// TwinCAT 3 PLC project Assembly_2_PLC
// ProgramVersion: 3.1.4022.7
// libraries:
//   Tc2_Standard, * (Beckhoff Automation GmbH)
//   Tc2_System, * (Beckhoff Automation GmbH)
//   Tc3_Module, * (Beckhoff Automation GmbH)
// project tree:
//   GVLs/ HMI.TcGVL
//   / PlcTask.TcTTO
//   POUs/00 System/ fbControl.TcPOU
//   POUs/01 Infeed/ fbInConveyor.TcPOU
//   POUs/02 Fitting/ fbHousingDelivery.TcPOU, fbInsertPlacing.TcPOU
//   POUs/03 Pressing/ fbHandling.TcPOU, fbPressing.TcPOU
//   POUs/ MAIN.TcPOU
// real-time tasks:
//   TASK PlcTask: cycle T#10ms, priority 20, ADS port 350
// I/O:
//   DEVICE Device 2 (EtherCAT), AmsNetId 10.133.61.48.3.1
//     Term 1 (EK1814) Console [EK1814 EtherCAT IO-Coupler  (0,5A E-Bus, 4 Ch. Dig. In, 3ms, 4 Ch. Dig. Out 24V, 0,5A)]
//       Term 2 (EL6900) FS Logic [EL6900, TwinSAFE PLC]
//       Term 3 (EL1904) FS DI1 [EL1904, 4 Ch. Safety Input 24V, TwinSAFE]
//         modules: Module 1 (FSOES)
//       Term 4 (EL1904) FS DI2 [EL1904, 4 Ch. Safety Input 24V, TwinSAFE]
//         modules: Module 1 (FSOES)
//       Term 5 (EL2904) FS DQ [EL2904, 4 Ch. Safety Output 24V, 0.5A, TwinSAFE]
//         modules: Module 1 (FSOES), Module 2 (DO)
//       Term 6 (EL1809) ST DI [EL1809 16Ch. Dig. Input 24V, 3ms]
//       Term 7 (EL2809) ST DQ [EL2809 16Ch. Dig. Output 24V, 0.5A]
//       Term 8 (EK1110) [EK1110 EtherCAT extension]
//     Term 9 (EK1100) Placing [EK1100 EtherCAT Coupler (2A E-Bus)]
//       Term 10 (EL1809) ST DI [EL1809 16Ch. Dig. Input 24V, 3ms]
//       Term 11 (EL2809) ST DQ [EL2809 16Ch. Dig. Output 24V, 0.5A]
//       Term 23 (EL9011) [EL9011 End Terminal]
//     Term 12 (EK1100) Pressing [EK1100 EtherCAT Coupler (2A E-Bus)]
//       Term 13 (EL1809) ST DI [EL1809 16Ch. Dig. Input 24V, 3ms]
//       Term 14 (EL2809) ST DQ [EL2809 16Ch. Dig. Output 24V, 0.5A]
//       Term 15 (EL3102) ST AI [EL3102 2Ch. Ana. Input +/-10V, Diff.]
//       Term 16 (EL4032) ST AQ [EL4032 2Ch. Ana. Output +/-10V, 12bit]
//       Term 24 (EL9011) [EL9011 End Terminal]
//     Term 17 (EK1100) External [EK1100 EtherCAT Coupler (2A E-Bus)]
//       Term 18 (EL1904) FS DI1 [EL1904, 4 Ch. Safety Input 24V, TwinSAFE]
//         modules: Module 1 (FSOES)
//       Term 19 (EL1904) FS DI2 [EL1904, 4 Ch. Safety Input 24V, TwinSAFE]
//         modules: Module 1 (FSOES)
//       Term 20 (EL2904) FS DQ [EL2904, 4 Ch. Safety Output 24V, 0.5A, TwinSAFE]
//         modules: Module 1 (FSOES), Module 2 (DO)
//       Term 21 (EL1808) ST DI [EL1808 8Ch. Dig. Input 24V, 3ms]
//       Term 22 (EL2808) ST DQ [EL2808 8Ch. Dig. Output 24V, 0.5A]
//       Term 25 (EL9011) [EL9011 End Terminal]
// variable links:
//   Device 2 (EtherCAT) <-> Device 2 (EtherCAT)/Term 1 (EK1814) Console/Term 2 (EL6900) FS Logic
//     Term 1 (EK1814) Console/Term 3 (EL1904) FS DI1/Module 1 (FSOES)/RxPDO/FSOE <-> ConnectionInputs/Message_2 TxPDO
//     Term 1 (EK1814) Console/Term 3 (EL1904) FS DI1/Module 1 (FSOES)/TxPDO/FSOE <-> ConnectionOutputs/Message_2 RxPDO
//     Term 1 (EK1814) Console/Term 5 (EL2904) FS DQ/Module 1 (FSOES)/TxPDO/FSOE <-> ConnectionOutputs/Message_4 RxPDO
//     Term 17 (EK1100) External/Term 20 (EL2904) FS DQ/Module 1 (FSOES)/RxPDO/FSOE <-> ConnectionInputs/Message_7 TxPDO
//     Term 17 (EK1100) External/Term 20 (EL2904) FS DQ/Module 1 (FSOES)/TxPDO/FSOE <-> ConnectionOutputs/Message_7 RxPDO
//   Device 2 (EtherCAT) <-> Device 2 (EtherCAT)/Term 1 (EK1814) Console/Term 4 (EL1904) FS DI2
//     Term 1 (EK1814) Console/Term 2 (EL6900) FS Logic/ConnectionInputs/Message_3 TxPDO <-> Module 1 (FSOES)/RxPDO/FSOE
//     Term 1 (EK1814) Console/Term 2 (EL6900) FS Logic/ConnectionOutputs/Message_3 RxPDO <-> Module 1 (FSOES)/TxPDO/FSOE
//   Device 2 (EtherCAT) <-> Device 2 (EtherCAT)/Term 1 (EK1814) Console/Term 5 (EL2904) FS DQ
//     Term 1 (EK1814) Console/Term 2 (EL6900) FS Logic/ConnectionInputs/Message_4 TxPDO <-> Module 1 (FSOES)/RxPDO/FSOE
//   Assembly_2_PLC/Assembly_2_PLC Instance <-> Device 2 (EtherCAT)/Term 1 (EK1814) Console/Term 2 (EL6900) FS Logic
//     PlcTask Inputs/MAIN.estopPressed <-> StandardInputs/Standard Out Var 9
//     PlcTask Inputs/MAIN.systemOk <-> StandardInputs/Standard Out Var 10
//     PlcTask Outputs/MAIN.doorUnlock_But <-> StandardOutputs/Standard In Var 8
//     PlcTask Outputs/MAIN.safeGroupErrorReset <-> StandardOutputs/Standard In Var 1

CONFIGURATION Assembly_2_PLC
    RESOURCE PLC ON TwinCAT3
        TASK PlcTask(INTERVAL := T#10ms, PRIORITY := 20);
        PROGRAM MAIN WITH PlcTask : MAIN;
    END_RESOURCE
END_CONFIGURATION

// ---- GVLs/HMI.TcGVL
{attribute 'qualified_only'}
VAR_GLOBAL

	DoorUnlockCmd	: BOOL;
	
END_VAR

// ---- POUs/MAIN.TcPOU
PROGRAM MAIN
VAR
	systemOk				AT %I* :BOOL;
	estopPressed			AT %I* :BOOL;
	safeGroupErrorReset  	AT %Q* :BOOL;
	doorUnlock_But		 	AT %Q* :BOOL;	
	
	SafetyResetPulse				: TP;
	
	Control							: fbControl;
	InfeedConveyor					: fbInConveyor;
	HousingDelivery					: fbHousingDelivery;
	InsertPlacing					: fbInsertPlacing;
	Handling						: fbHandling;
	Pressing						: fbPressing;
	
END_VAR

doorUnlock_But := HMI.DoorUnlockCmd;
//gpb.estopOk := systemOk;

//===============================================================================================
// Safety reset at system startup
//===============================================================================================
SafetyResetPulse(IN:=TRUE, PT:= T#500MS , Q=>safeGroupErrorReset , ET=> );



//===============================================================================================
// Machine modes and status indication 
//===============================================================================================

Control(
	SafetyOk:= SystemOk,
	ResetCompleted := TRUE,
	ResetCmd=> , 
	AutoCycle=> , 
	ManualMode=> , 
	DoorUnlockCmd=> );

//===============================================================================================
// Infeed conveyor control  
//===============================================================================================

InfeedConveyor(
	SafetyOk:= , 
	ResetCmd:= , 
	AutoCycle:= , 
	ManualCmd:= , 
	ResetCompleted=> );


	
	
//===============================================================================================
// Fitting station process control  
//===============================================================================================

HousingDelivery(
	SafetyOk:= , 
	ResetCmd:= , 
	AutoCycle:= , 
	ManualCmd:= , 
	ResetCompleted=> );
	
InsertPlacing(
	SafetyOk:= , 
	ResetCmd:= , 
	AutoCycle:= , 
	ManualCmd:= , 
	ResetCompleted=> );	

	
//===============================================================================================
// Pressing station process control  
//===============================================================================================	


Handling(
	SafetyOk:= , 
	ResetCmd:= , 
	AutoCycle:= , 
	ManualCmd:= , 
	ResetCompleted=> );


Pressing(
	SafetyOk:= , 
	ResetCmd:= , 
	AutoCycle:= , 
	ManualCmd:= , 
	ResetCompleted=> );

END_PROGRAM

// ---- POUs/00 System/fbControl.TcPOU
FUNCTION_BLOCK fbControl
VAR_INPUT
	SafetyOk			: BOOL;
	ServosEnable		: BOOL;
	ResetCompleted		: BOOL;
END_VAR
VAR_OUTPUT
	ResetCmd				: BOOL;
	AutoCycle 				: BOOL;
	ManualMode				: BOOL;
	DoorUnlockCmd			: BOOL;
	
END_VAR
VAR
	// Operator Console	
	StartPB				AT%I* : BOOL;
	StopPB				AT%I* : BOOL;
	ManualKeySW			AT%I* : BOOL;
	ResetPB				AT%I* : BOOL;
	DoorUnlockPB		AT%I* : BOOL;
	StartIndicator		AT%Q* : BOOL;
	ResetIndicator		AT%Q* : BOOL;
	Q1Indicator			AT%Q* : BOOL;
	Q2Indicator			AT%Q* : BOOL;
	
	// Signal tower
	RedTower			AT%Q* : BOOL;
	YellowTower			AT%Q* : BOOL;
	GreenTower			AT%Q* : BOOL;
	
	PulseONTime			  		: TON;
	PulseOFFTime			  	: TON;
	ClockPulse					: BOOL;
		
	State 						: INT := 0;

END_VAR


//===============================================================================================
// State machine 
//===============================================================================================

CASE State OF
	
0: // Estop 
	ManualMode := 0;
	ResetCmd := 0;
	AutoCycle := 0;
	
	IF SafetyOk THEN
		State := 1;
	END_IF
	
	
	
1: 	// Automatic mode. Wait for Reset initiation.
	// Allow switching to Manual mode.
	ManualMode := 0;
	ResetCmd := 0;
	AutoCycle := 0;
	
	// Auto mode selected. Wait for reset/homing to be requested.
	IF NOT ManualKeySW AND ResetPB THEN
		State := 2;
	END_IF
	
	// Manual mode selected
	IF ManualKeySW THEN
		State := 5;
	END_IF


2: 	// Automatic mode. Reset/homing requested. 
	ResetCmd := 1;
	
	//Waiting for confirmation.
	IF ResetCompleted THEN
		State := 3;
	END_IF


3:	// Automatic mode. Wait for Automatic cycle request or Manual mode request. 	
	ResetCmd := 0;
	AutoCycle := 0;
	
	IF NOT ManualKeySW AND StartPB THEN
		State := 4;
	END_IF
		
	IF ManualKeySW THEN
		State := 5;
	END_IF
	
4: // Auto cycle activated
	AutoCycle := 1;
	
	IF NOT StopPB THEN
		State := 3;
	END_IF

5: // Manual mode
	ManualMode := 1;

	IF NOT ManualKeySW THEN
		State := 1;
	END_IF
	
END_CASE

// Switch to initial state when Emergency stop has been activated.
IF NOT SafetyOk THEN
	State := 0;
END_IF



//===============================================================================================
// Clock pulse
//===============================================================================================
PulseONTime(IN:= NOT PulseOFFTime.Q, PT:= T#500MS, Q=> ClockPulse, ET=> );
PulseOFFTime(IN:= PulseONTime.Q, PT:= T#500MS, Q=> , ET=> );





//===============================================================================================
// Physical outputs - Operator console
//===============================================================================================

// Reset PB indicator flashes when the machine requires reset/homing.
// It is ON solid when the machine homing is in progress, and OFF in all other states of the system.
ResetIndicator := State = 1 AND ClockPulse OR  State = 2;


// Start PB indicator flashes when the machine is ready for the workcycle to be started.
// It is ON solid when machine workcycle is in progress and OFF in all other states of the system.
StartIndicator := State = 3 AND ClockPulse OR State = 4;


// Console indicator 1 is ON solid when Servo Enable is activated.
Q1Indicator := ServosEnable;

// Console indicator 2 is ON solid when Manual is activated.
// Console indicator 2 flashes when manual keyswitch is switched to manual during autocycle
Q2Indicator := State = 1 AND ClockPulse OR State = 5;






//===============================================================================================
// Physical outputs - Signal tower
//===============================================================================================

// Red signal tower is ON solid when safety is not activated
//RedTower := State = 0 OR State = 5 AND ClockPulse;


// Yellow signal tower is ON solid when the machine is ready to start preparation for starting and when preparation has been completed.
// Yellow signal tower flashes when homing/reset is in progress
//YellowTower :=  State = 1 OR State = 2 AND ClockPulse OR state = 3;

// Green signal tower is ON when Auto Cycle is activated
//GreenTower := State = 4;

END_FUNCTION_BLOCK

// ---- POUs/01 Infeed/fbInConveyor.TcPOU
FUNCTION_BLOCK fbInConveyor
VAR_INPUT
	SafetyOk			: BOOL;
	ResetCmd			: BOOL;
	AutoCycle			: BOOL;
	ManualCmd			: BOOL;
	
END_VAR
VAR_OUTPUT
	ResetCompleted 		: BOOL;
	
END_VAR
VAR
	FwdConveyor			AT %Q* :BOOL;
	State						: INT := 0;
END_VAR

END_FUNCTION_BLOCK

// ---- POUs/02 Fitting/fbHousingDelivery.TcPOU
FUNCTION_BLOCK fbHousingDelivery
VAR_INPUT
	SafetyOk			: BOOL;
	ResetCmd			: BOOL;
	AutoCycle			: BOOL;
	ManualCmd			: BOOL;
END_VAR
VAR_OUTPUT
	ResetCompleted 		: BOOL;
	
END_VAR
VAR
	

	WpAtStart			AT %I* :BOOL;
	WpAtPlacing			AT %I* :BOOL;
	
	FwdConveyor			AT %Q* :BOOL;
	AdvanceGate1		AT %Q* :BOOL;
	RetractGate2		AT %Q* :BOOL;
	
	State				: INT := 0;

END_VAR

END_FUNCTION_BLOCK

// ---- POUs/02 Fitting/fbInsertPlacing.TcPOU
FUNCTION_BLOCK fbInsertPlacing
VAR_INPUT
	SafetyOk			: BOOL;
	ResetCmd			: BOOL;
	AutoCycle			: BOOL;
	ManualCmd			: BOOL;
	
END_VAR
VAR_OUTPUT
	ResetCompleted 		: BOOL;
	
END_VAR
VAR
	
	WpAvailable			AT %I* :BOOL;
	WpVacGripped		AT %I* :BOOL;
	SlideYRetracted		AT %I* :BOOL;
	SlideYExtended		AT %I* :BOOL;
	SlideZUp			AT %I* :BOOL;
	
	
	AdvanceSlideY		AT %Q* :BOOL;
	RetractSlideY		AT %Q* :BOOL;
	LowerSlideZ			AT %Q* :BOOL;
	VacuumOn			AT %Q* :BOOL;
	
	State				: INT := 0;

END_VAR

END_FUNCTION_BLOCK

// ---- POUs/03 Pressing/fbHandling.TcPOU
FUNCTION_BLOCK fbHandling
VAR_INPUT
	SafetyOk			: BOOL;
	ResetCmd			: BOOL;
	AutoCycle			: BOOL;
	ManualCmd			: BOOL;
	
END_VAR
VAR_OUTPUT
	ResetCompleted 		: BOOL;
	
END_VAR
VAR
	WpInGripper				AT %I* :BOOL;
	LinearAtCentre			AT %I* :BOOL;
	LinearAtExit			AT %I* :BOOL;
	RotaryAtPickup			AT %I* :BOOL;
	RotaryAtPress			AT %I* :BOOL;
	RotaryAtDropoff			AT %I* :BOOL;

	CloseGripper			AT %Q* :BOOL;
	LinearToExit			AT %Q* :BOOL;
	LinearToCentre			AT %Q* :BOOL;
	RotaryToPickup			AT %Q* :BOOL;
	RotaryToPress			AT %Q* :BOOL;
	RotaryToDropoff			AT %Q* :BOOL;
	
	
	State				: INT := 0;

END_VAR

END_FUNCTION_BLOCK

// ---- POUs/03 Pressing/fbPressing.TcPOU
FUNCTION_BLOCK fbPressing
VAR_INPUT
	SafetyOk			: BOOL;
	ResetCmd			: BOOL;
	AutoCycle			: BOOL;
	ManualCmd			: BOOL;
END_VAR
VAR_OUTPUT
	ResetCompleted 		: BOOL;
		
END_VAR
VAR
	
	ForceReached			AT %I* :BOOL;
	
	AdvancePress			AT %Q* :BOOL;
	
	State					: INT := 0;

END_VAR

END_FUNCTION_BLOCK
